(* CoDeSys 2.3 export: FGETK15PUMP.EXP *)

(* POU K15/fGetK15Pump, ST *)
FUNCTION fGetK15Pump :BOOL
(* Проверка включения насоса*)
VAR_INPUT
	PumpID : USINT;
END_VAR
fGetK15Pump := PLC160DO.K15Pump[PumpID];
END_FUNCTION
